{attribute 'GeneratedUsingTerminal: EK1100-0000-0018'}
{attribute addProperty BoxType "EK1100-0000-0018"}
{attribute addProperty Id "Beckhoff_ER2xxxEK1122Beckhoff_ER2xxxEK1122_E7B52A1E904"}
{attribute addProperty CRC "3700805188"}
{attribute addProperty Size "904"}
TYPE Beckhoff_ER2xxx_DC95CE44 EXTENDS EK1100_1FC0878B :
STRUCT
	{attribute addProperty Name "Beckhoff_ER2xxxEK1122"}
	{attribute addProperty PreviousPort "Beckhoff ER2xxx : B"}
	Beckhoff_ER2xxxEK1122 : Beckhoff_ER2xxxEK1122_E7B52A1E;
END_STRUCT
END_TYPE

(* stored: Version 1.2.0.0, ProductVersion 3.1.4024.9
   DUT Beckhoff_ER2xxx_DC95CE44: Id {8f90ba54-1895-4c75-8532-084e65cf5b5e} *)
